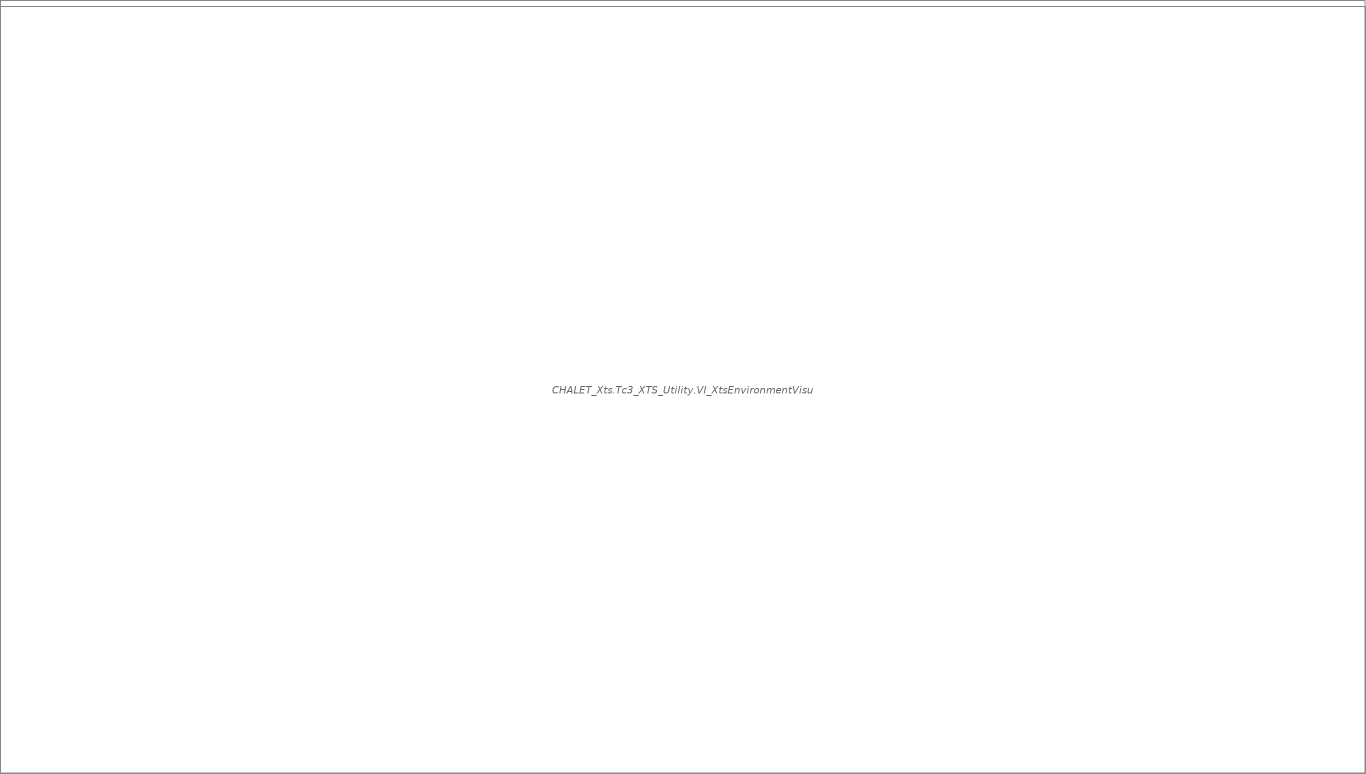
VISUALIZATION Visualization  // 1366x774
    Frame (0,6 1366x768)
        shows CHALET_Xts.Tc3_XTS_Utility.VI_XtsEnvironmentVisu()
END_VISUALIZATION

(* stored: Version 1.1.0.1, ProductVersion 3.1.4024.12
   Visu Visualization: Id {b4a227ed-af87-4a41-b751-d639d99f2160} *)
